# B&R Automation Studio project BasePLC
Automation Studio 4.7.2.98

## Configuration Config1

### Hardware
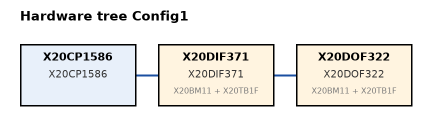
```
X20BM11 : X20BM11 v1.0.0.1  [X2X1 -> X20CP1586.IF6]
X20BM11a : X20BM11 v1.0.0.1  [X2X1 -> X20BM11.X2X2]
X20CP1586 : X20CP1586 v1.8.0.0
  Connector IF2:
    ActivateDevice = 1
    Mode = Manual
    InternetAddress = 192.168.10.10
    SubnetMask = 255.255.255.0
  ConfigurationID = youtube_Config1
X20DIF371 : X20DIF371 v1.1.0.0  [SS1 -> X20TB1F.SS; SL -> X20BM11.SL1]
X20DOF322 : X20DOF322 v1.3.0.0  [SS1 -> X20TB1F1.SS; SL -> X20BM11a.SL1]
X20TB1F : X20TB1F v1.0.0.0
X20TB1F1 : X20TB1F v1.0.0.0
```

### IoMap.iom - X20CP1586/IoMap.iom
```iecst
VAR_CONFIG
	::Program:Test AT %QX."X20DOF322".DigitalOutput01;
END_VAR
```

## Logical view

### Program Logical/Program

#### Variables.var
```iecst
VAR
	Test : BOOL;
END_VAR
```

#### Main.c
```c
#include <bur/plctypes.h>

#ifdef _DEFAULT_INCLUDES
	#include <AsDefault.h>
#endif

void _INIT ProgramInit(void)
{
	Test = 1;
}

void _CYCLIC ProgramCyclic(void)
{
	if (Test == 1)
		Test = 0;
	else
		Test = 1;
}

void _EXIT ProgramExit(void)
{

}
```
